TYPE ST_AxisData :
STRUCT
    fActPosition : LREAL;
    fSetPosition : LREAL;
    fActVelocity : LREAL;
    fSetVelocity : LREAL;
    fPositionDiff: LREAL;
    fActRpm      : LREAL;
    fActTorque   : LREAL;
END_STRUCT
END_TYPE

(* stored: Version 1.1.0.1, ProductVersion 3.1.4026.18
   DUT ST_AxisData: Id {bf71d3e8-0d5d-433d-bc31-6a2106ce1b99} *)
